TYPE EP7402_REF :
STRUCT
	stInputs	AT %I* : ARRAY[0..7] OF BYTE;//MDR_CONTROL.EP7402_Inputs;
	stOutputs	AT %Q* : ARRAY[0..7] OF BYTE;//MDR_Control.EP7402_Outputs;
END_STRUCT
END_TYPE

(* stored: Version 1.1.0.1, ProductVersion 3.1.4024.11
   DUT EP7402_REF: Id {e41a4876-ed96-4689-861d-e491bef68390} *)
